// TIA Portal V17 export
// export: Created 2025-07-13T07:36:02.8341503Z, ExportSetting WithDefaults, DisplayName Totally Integrated Automation Portal, DisplayVersion V17, DisplayName TIA Portal Openness, DisplayVersion V17, DisplayName TIA Portal Version Control Interface, DisplayVersion V17, DisplayName STEP 7 Professional, DisplayVersion V17, DisplayName STEP 7 Safety, DisplayVersion V17, DisplayName WinCC Advanced / Unified PC, DisplayVersion V17
FUNCTION "pump_action" : Void   // FC1, LAD
{ S7_Optimized_Access := 'TRUE' }
VERSION : 0.1
// stored: AutoNumber true, IsIECCheckEnabled false, SetENOAutomatically false, UDAEnableTagReadback false
BEGIN

REGION Network 1
   // 1号泵
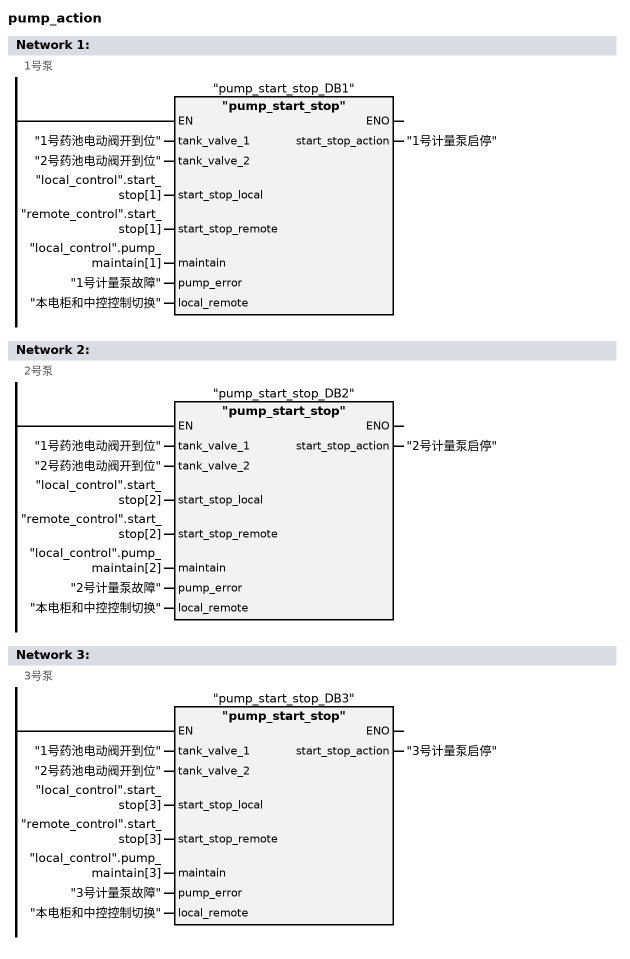
   RUNG wire#powerrail
      "pump_start_stop_DB1"(tank_valve_1 := "1号药池电动阀开到位", tank_valve_2 := "2号药池电动阀开到位", start_stop_local := "local_control".start_stop[1], start_stop_remote := "remote_control".start_stop[1], maintain := "local_control".pump_maintain[1], pump_error := "1号计量泵故障", local_remote := "本电柜和中控控制切换", start_stop_action => "1号计量泵启停")
   END_RUNG
   // the same network as SCL:
   "pump_start_stop_DB1"(tank_valve_1 := "1号药池电动阀开到位",   // "pump_start_stop"
                         tank_valve_2 := "2号药池电动阀开到位",
                         start_stop_local := "local_control".start_stop[1],
                         start_stop_remote := "remote_control".start_stop[1],
                         maintain := "local_control".pump_maintain[1],
                         pump_error := "1号计量泵故障",
                         local_remote := "本电柜和中控控制切换",
                         start_stop_action => "1号计量泵启停");
END_REGION

REGION Network 2
   // 2号泵
   RUNG wire#powerrail
      "pump_start_stop_DB2"(tank_valve_1 := "1号药池电动阀开到位", tank_valve_2 := "2号药池电动阀开到位", start_stop_local := "local_control".start_stop[2], start_stop_remote := "remote_control".start_stop[2], maintain := "local_control".pump_maintain[2], pump_error := "2号计量泵故障", local_remote := "本电柜和中控控制切换", start_stop_action => "2号计量泵启停")
   END_RUNG
   // the same network as SCL:
   "pump_start_stop_DB2"(tank_valve_1 := "1号药池电动阀开到位",   // "pump_start_stop"
                         tank_valve_2 := "2号药池电动阀开到位",
                         start_stop_local := "local_control".start_stop[2],
                         start_stop_remote := "remote_control".start_stop[2],
                         maintain := "local_control".pump_maintain[2],
                         pump_error := "2号计量泵故障",
                         local_remote := "本电柜和中控控制切换",
                         start_stop_action => "2号计量泵启停");
END_REGION

REGION Network 3
   // 3号泵
   RUNG wire#powerrail
      "pump_start_stop_DB3"(tank_valve_1 := "1号药池电动阀开到位", tank_valve_2 := "2号药池电动阀开到位", start_stop_local := "local_control".start_stop[3], start_stop_remote := "remote_control".start_stop[3], maintain := "local_control".pump_maintain[3], pump_error := "3号计量泵故障", local_remote := "本电柜和中控控制切换", start_stop_action => "3号计量泵启停")
   END_RUNG
   // the same network as SCL:
   "pump_start_stop_DB3"(tank_valve_1 := "1号药池电动阀开到位",   // "pump_start_stop"
                         tank_valve_2 := "2号药池电动阀开到位",
                         start_stop_local := "local_control".start_stop[3],
                         start_stop_remote := "remote_control".start_stop[3],
                         maintain := "local_control".pump_maintain[3],
                         pump_error := "3号计量泵故障",
                         local_remote := "本电柜和中控控制切换",
                         start_stop_action => "3号计量泵启停");
END_REGION
END_FUNCTION
